FUNCTION_BLOCK FB_EtherCATBus EXTENDS FB_ComponentBase

VAR
	/// IO structure
	stIO 				: REFERENCE TO ST_EtherCatIO;
	oldEtherCATState	: INT;
	n3072Err			: INT;
END_VAR

///
/// EtherCAT driver.
/// Hannes Fuger / asma.at / 12.2015
///

METHOD FB_init : BOOL
VAR_INPUT
	bInitRetains : BOOL; // if TRUE, the retain variables are initialized (warm start / cold start)
	bInCopyCode : BOOL;  // if TRUE, the instance afterwards gets moved into the copy code (online change)
END_VAR
eTyp := E_ComponentType.eComponentType_EtherCAT;
END_METHOD

METHOD Run : E_ComponentState
VAR_INPUT
END_VAR
// base logic run
Run := SUPER^.Run();

// chk reference
IF NOT __ISVALIDREF(fbEventLog) THEN
	RETURN;
END_IF

IF oldEtherCATState = stIo.eEtherCATState THEN
	RETURN;
ELSE
	oldEtherCATState := stIo.eEtherCATState;
END_IF



// switch EtherCAT State
CASE stIO.eEtherCATState OF
	/// Link error
	eEtherCATState_LinkError :
		WriteError(eEvent_hardwareError, 'EtherCAT: Link error');
		
	/// I/O locked after link error (I/O reset required)
	eEtherCATState_IoLockedAfterLinkErr :
		WriteError(eEvent_hardwareError, 'EtherCAT: I/O locked after link error (I/O reset required)');
	
	/// Link error (redundancy adapter)
	eEtherCATState_LinkErrRedAdapter :
		WriteError(eEvent_hardwareError, 'EtherCAT: Link error (redundancy adapter)');
	
	/// Missing one frame (redundancy mode)
	eEtherCATState_MissingFrame :
		WriteError(eEvent_hardwareError, 'EtherCAT: Missing one frame (redundancy mode)');
	
	/// Out of send resources (I/O reset required)
	eEtherCATState_OutOfSendResources :
		WriteError(eEvent_hardwareError, 'EtherCAT: Out of send resources (I/O reset required)');
	
	/// Watchdog triggered
	eEtherCATState_WatchdogTriggered :
		WriteError(eEvent_hardwareError, 'EtherCAT: Watchdog triggered');
	
	/// Ethernet driver (miniport) not found
	eEtherCATState_EthernetDrvNotFound :
		WriteError(eEvent_hardwareError, 'EtherCAT: Ethernet driver (miniport) not found');
	
	/// I/O reset active
	eEtherCATState_IO_resetActive :
		WriteError(eEvent_hardwareError, 'EtherCAT: I/O reset active');
	
	/// At least one device in 'INIT' state
	eEtherCATState_AtLeastOneDeviceInit :
		WriteError(eEvent_hardwareError, 'EtherCAT: At least one device in INIT state');
	
	///  At least one device in 'PRE-OP' state
	eEtherCATState_AtLeastOneDevicePreOp :
		WriteError(eEvent_hardwareError, 'EtherCAT: At least one device in PRE-OP state');
	
	/// At least one device in 'SAFE-OP' state
	eEtherCATState_AtLeastOneDeviceSafeOp :
		WriteError(eEvent_hardwareError, 'EtherCAT: At least one device in SAFE-OP state');
	
	/// At least one device indicates an error state
	eEtherCATState_AtLeastOneDeviceError :
		WriteError(eEvent_hardwareError, 'EtherCAT: At least one device indicates an error state');
	
	/// DC not in sync
	eEtherCATState_DC_notInSync :
		WriteError(eEvent_hardwareError, 'EtherCAT: DC not in sync');

	ELSE // default 
		IF stIO.eEtherCATState = 1024 THEN
			n3072Err := n3072Err + 1;
		ELSIF stIO.eEtherCATState = 3072 THEN
			n3072Err := n3072Err + 1;
		ELSIF stIO.eEtherCATState <> 0 THEN
			WriteError(eEvent_hardwareError, Concat('EtherCAT Error: ', INT_TO_STRING(stIO.eEtherCATState)));
		END_IF
	
END_CASE
END_METHOD

/// Dependency injection method.
{attribute 'object_name' := 'SetReferences'}
METHOD SetReferences
VAR_IN_OUT
	/// IO structure
	stRefIO		: ST_EtherCatIO;
END_VAR
/// set up references
stIO REF= stRefIO;
END_METHOD

END_FUNCTION_BLOCK

(* stored: Version 1.1.0.1, ProductVersion 3.1.4022.9
   POU FB_EtherCATBus: Id {55f2b2ae-663d-494c-86e1-ccb5cb9949fd}, SpecialFunc None
   Method FB_init: Id {29a3bf8c-a6c8-4ef7-99a3-f5067604e32f}
   Method Run: Id {3e887635-f8de-4acc-be05-4b1be9527b99}
   Method SetReferences: Id {87c0e814-fac0-455c-a362-eecf97c34742} *)
